// TwinCAT 3 PLC project MicroTestStandPPM
// ProgramVersion: 3.1.4020.5
// libraries:
//   lcls-twincat-motion-zlentz, * (SLAC)
//   lcls2-cc-lib-zlentz, * (SLAC)
//   Tc2_Standard, * (Beckhoff Automation GmbH)
//   Tc2_System, * (Beckhoff Automation GmbH)
//   Tc2_Utilities, * (Beckhoff Automation GmbH)
//   Tc3_Module, * (Beckhoff Automation GmbH)
// project tree:
//   / PlcTask.TcTTO
//   POUs/ Main.TcPOU
// real-time tasks:
//   TASK PlcTask: cycle T#1ms, priority 20, ADS port 350
// motion (NC):
// I/O:
//   DEVICE Device 1 (EtherCAT), AmsNetId 172.21.148.185.2.1
//     Term 1 (EK1200) [EK1200-5000 EtherCAT Power supply (2A E-Bus)]
//       Term 2 (EL6695) [EL6695 EtherCAT Bridge terminal (Primary)]
//       Term 3 (EK1110) [EK1110 EtherCAT extension]
//     Term 4 (EK1100) [EK1100 EtherCAT Coupler (2A E-Bus)]
//       Term 5 (EL7041) [EL7041 1Ch. Stepper motor output stage (50V, 5A)]
//       Term 6 (EL5042) [EL5042 2Ch. BiSS-C Encoder]
//       Term 7 (EL2004) [EL2004 4Ch. Dig. Output 24V, 0.5A]
//       Term 8 (EL3314) [EL3314 4Ch. Ana. Input Thermocouple (TC)]
//       Term 9 (EL3052) [EL3052 2Ch. Ana. Input 4-20mA]
//       Term 10 (EL3062) [EL3062 2Ch. Ana. Input 0-10V]
//       Term 11 (EL4004) [EL4004 4Ch. Ana. Output 0-10V, 12bit]
//       Term 12 (EL9011) [EL9011 End Terminal]
// variable links:
//   MicroTestStandPPM Instance <-> Device 1 (EtherCAT)/Term 4 (EK1100)/Term 10 (EL3062)
//     PlcTask Inputs/Main.fbPPM.stPPM.stPowerMeter.iVoltageINT <-> AI Standard Channel 1/Value
//   MicroTestStandPPM Instance <-> Device 1 (EtherCAT)/Term 4 (EK1100)/Term 11 (EL4004)
//     PlcTask Outputs/Main.fbPPM.stPPM.stGige.iIlluminatorINT <-> AO Outputs Channel 1/Analog output
//   MicroTestStandPPM Instance <-> Device 1 (EtherCAT)/Term 4 (EK1100)/Term 5 (EL7041)
//     PlcTask Inputs/Main.M1.bLimitBackwardEnable <-> STM Status/Status/Digital input 2
//     PlcTask Inputs/Main.M1.bLimitForwardEnable <-> STM Status/Status/Digital input 1
//   MicroTestStandPPM Instance <-> Device 1 (EtherCAT)/Term 4 (EK1100)/Term 7 (EL2004)
//     PlcTask Outputs/Main.M1.bBrakeRelease <-> Channel 1/Output
//     PlcTask Outputs/Main.fbPPM.stPPM.stGige.bGigePower <-> Channel 2/Output
//   MicroTestStandPPM Instance <-> Device 1 (EtherCAT)/Term 4 (EK1100)/Term 8 (EL3314)
//     PlcTask Inputs/Main.fbPPM.stPPM.fYagThermoCouple <-> TC Inputs Channel 2/Value
//     PlcTask Inputs/Main.fbPPM.stPPM.stPowerMeter.fThermoCouple <-> TC Inputs Channel 1/Value
//   MicroTestStandPPM Instance <-> NC-Task 1 SAF/Axes/MMS_Y
//     PlcTask Inputs/Main.M1.Axis.NcToPlc <-> Outputs/ToPlc
//     PlcTask Outputs/Main.M1.Axis.PlcToNc <-> Inputs/FromPlc

CONFIGURATION MicroTestStandPPM
    RESOURCE PLC ON TwinCAT3
        TASK PlcTask(INTERVAL := T#1ms, PRIORITY := 20);
        PROGRAM Main WITH PlcTask : Main;
    END_RESOURCE
END_CONFIGURATION

// ---- POUs/Main.TcPOU
PROGRAM Main
VAR
	{attribute 'pytmc' := '
        pv: TST:PPM:MMS:Y
	'}
	M1: DUT_MotionStage;
	
	{attribute 'pytmc' := '
		pv: TST
	'}
	fbPPM: FB_PPM;
END_VAR

fbPPM(stYStage := M1);

END_PROGRAM
